Universal Robots PolyScope program: programa.urp

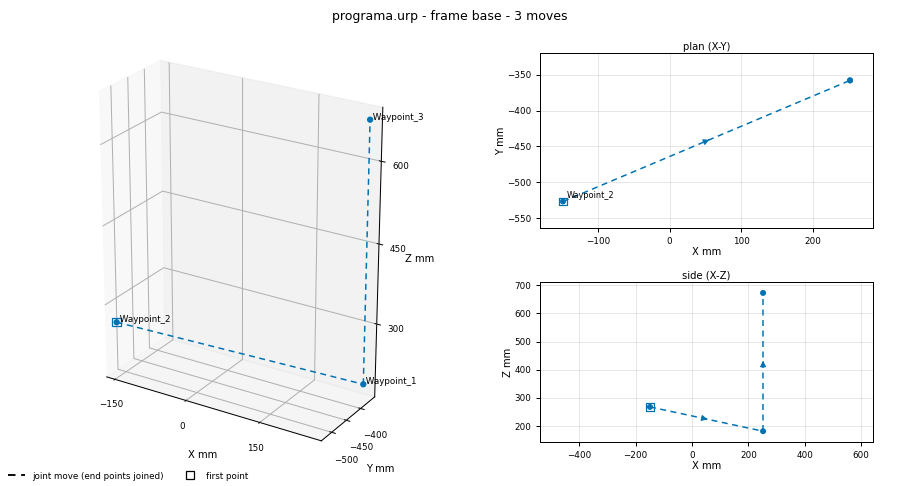
[picture p0: tool path of programa.urp in frame base, 3 of 3 moves have a stored position in this frame; points joined in program order, loops and branches not executed]
Program programa (installation=default directory=/ursim/programs/programs.UR5 createdIn=5.4.2.76197 lastSavedIn=5.4.2.76197 robotSerialNumber=20183599999)
Calibrated DH parameters: a=[0, -0.425, -0.3922, 0, 0, 0]; d=[0.1625, 0, 0, 0.1333, 0.0997, 0.0996]; alpha=[1.570796, 0, 0, 1.570796, -1.570796, 0]; deltaTheta=[0, 0, 0, 0, 0, 0]
Robot Program (runOnlyOnce=false)
  Loop Forever
    MoveJ speed 60 deg/s, acceleration 80 deg/s^2 (useActiveTCP=true) feature=Base
      Waypoint Waypoint_2: TCP in base x=-148.946 y=-526.841 z=268.286 mm, rx=0.0041 ry=3.0988 rz=-0.3592 rad; joints [-92.012, -103.202, -113.387, -40.233, 91.695, -1.666] deg
    MoveJ speed 60 deg/s, acceleration 80 deg/s^2 (useActiveTCP=true) feature=Base
      Waypoint Waypoint_1: TCP in base x=252.169 y=-357.631 z=182.145 mm, rx=0.0112 ry=2.882 rz=-0.9643 rad; joints [-30.517, -104.55, -140.743, 1.258, 62.013, 53.351] deg
    If read_port_register(7)≟7
      MoveJ speed 60 deg/s, acceleration 80 deg/s^2 (useActiveTCP=true) feature=Base
        Waypoint Waypoint_3: TCP in base x=252.169 y=-357.631 z=672.428 mm, rx=0.0041 ry=3.0988 rz=-0.3592 rad; joints [-34.651, -82.471, -71.752, -107.141, 79.866, 54.733] deg
